// SIMATIC S7-200 project (STEP 7-Micro/WIN), CPU 224XP REL 02.00

ORGANIZATION_BLOCK 主:OB1
TITLE=程序注解
BEGIN
Network 1 // 网络标题
// 网络注解
LD     SM0.0
CALL   PID0_INIT:SBR2, AIW0, 80.0, VW200 //PID初始化，PID输出在VW200中
Network 2
LD     SM0.0
CALL   PWM0_RUN:SBR3, SM0.0, 32000, VW200, VB202 //Q0.0输出PWM脉冲
Network 3
LD     I1.0
A      SM0.5                 //SM0.5产生周期为1s的时钟脉冲      
EU                           //上升沿检测
MOVW   AIW0, 过程变量:VW130      //过程变量送数据归档缓冲区
MOVW   VW200, PID输出:VW132    //PID输出量送数据归档缓冲区
CALL   DAT0_WRITE:SBR1, VB21 //将过程变量和PID输出写入存储卡
END_ORGANIZATION_BLOCK

// SBR1: protected block, not included

// SBR2: protected block, not included

// SBR3: protected block, not included

// INT1: protected block, not included

// (further data pages could not be read)
